FUNCTION_BLOCK FB_SterowanieMaszyna
VAR_INPUT
END_VAR
VAR_OUTPUT
END_VAR
VAR
END_VAR

END_FUNCTION_BLOCK

(* stored: Version 1.1.0.1, ProductVersion 3.1.4024.11
   POU FB_SterowanieMaszyna: Id {13408bd3-8145-4c5f-8343-0c104b15fb7b}, SpecialFunc None *)
